// TIA Portal V16 export
// export: Created 2024-09-05T17:39:08.4487697Z, ExportSetting WithDefaults, DisplayName Totally Integrated Automation Portal, DisplayVersion V16 Update 6, DisplayName TIA Portal Version Control Interface, DisplayVersion V16 Update 2, DisplayName TIA Portal Openness, DisplayVersion V16 Update 6, DisplayName STEP 7 Professional, DisplayVersion V16 Update 6, DisplayName STEP 7 Safety, DisplayVersion V16, DisplayName WinCC Advanced, DisplayVersion V16 Update 6
DATA_BLOCK "SlidesMain_DB"   // DB45
VERSION : 0.1
// stored: AutoNumber true, DBAccessibleFromOPCUA true, InstanceOfName SlidesMain, InstanceOfType FB
"SlidesMain"
   // VAR
   //    R_TRIG_Instance { S7_SetPoint := 'True'} : R_TRIG;
   //    IEC_Timer_0_Instance { S7_SetPoint := 'True'} : TON_TIME;
   //    IEC_Timer_0_Instance_1 { S7_SetPoint := 'True'} : TOF_TIME;
   //    IEC_Timer_0_Instance_3 { S7_SetPoint := 'True'} : TON_TIME;
   //    IEC_Timer_0_Instance_5 { S7_SetPoint := 'True'} : TON_TIME;
   // END_VAR
BEGIN
   R_TRIG_Instance.CLK := FALSE;
   R_TRIG_Instance.Q := FALSE;
   R_TRIG_Instance.Stat_Bit := FALSE;
   IEC_Timer_0_Instance.PT := T#0MS;
   IEC_Timer_0_Instance.IN := FALSE;
   IEC_Timer_0_Instance_1.PT := T#0MS;
   IEC_Timer_0_Instance_1.IN := TRUE;
   IEC_Timer_0_Instance_3.PT := T#0MS;
   IEC_Timer_0_Instance_3.IN := FALSE;
   IEC_Timer_0_Instance_5.PT := T#0MS;
   IEC_Timer_0_Instance_5.IN := FALSE;
END_DATA_BLOCK
